VAR_GLOBAL
END_VAR

(* stored: Version 1.1.0.1, ProductVersion 3.1.0.23
   GVL CHD_CmdState: Id {c72de146-8b48-4304-9823-42d7c4fa5359} *)
